// TIA Portal project "Project1" (V19)

(* hardware
DEVICE "S7-1500/ET200MP station_1"  S7-1500 station
   slot 0: "Rail_0"  Rack  6ES7 590-1***0-0AA0
   slot 1: "PLC_1"  CPU 1513-1 PN  6ES7 513-1AL02-0AB0  V2.9
      slot 3: "CPU display_1"  6ES7591-1AA00-0AA0
      slot 32768: "PROFINET interface_1"  X1
         slot 32769: "Port_1"  X1 P1
         slot 32770: "Port_2"  X1 P2
      slot 34817: "Virtual CP interface port_1"  Virtual CP interface port  Virtual CP interface port
   slot 2: "DI 16x24VDC BA_1"  DI 16x24VDC BA  6ES7 521-1BH10-0AA0  V1.1
   slot 3: "DQ 16x24VDC/0.5A BA_1"  DQ 16x24VDC/0.5A BA  6ES7 522-1BH10-0AA0  V1.1
DEVICE "HMI_1"  KTP700 Basic PN
   slot 0: "HMI_1"  KTP700 Basic PN  6AV2 123-2GB03-0AX0  17.0.0.0
   slot 1: "HMI_RT_1"  KTP700 Basic PN  6AV2 123-2GB03-0AX0  17.0.0.0
   slot 5: "HMI_1.IE_CP_1"  PROFINET Interface  17.0.0.0
      slot 1: "PROFINET Interface_1"  PROFINET Interface
         slot 1: "Port_1"  Port
*)

// ===== PLC "PLC_1"  CPU 1513-1 PN =====

VAR_GLOBAL   // PLC tag table "Default tag table"
   "At Entry" AT %I0.0 : Bool;
   "At Load" AT %I0.1 : Bool;
   "At left" AT %I0.2 : Bool;
   "At Middle" AT %I0.3 : Bool;
   "At Right" AT %I0.4 : Bool;
   "At Unload" AT %I0.5 : Bool;
   "At Exit" AT %I0.6 : Bool;
   "Moving X" AT %I0.7 : Bool;
   "Moving Z" AT %I1.0 : Bool;
   "Start" AT %I1.1 : Bool;
   "Reset" AT %I1.2 : Bool;
   "Stop" AT %I1.3 : Bool;
   "Emergency stop" AT %I1.4 : Bool;
   "Auto" AT %I1.5 : Bool;
   "FACTORY I/O (Runing)" AT %I1.6 : Bool;
   "Entry Conveyor" AT %Q0.0 : Bool;
   "Load Conveyor" AT %Q0.1 : Bool;
   "Forks Left" AT %Q0.2 : Bool;
   "Forks Right" AT %Q0.3 : Bool;
   "Lift" AT %Q0.4 : Bool;
   "Unload Conveyor" AT %Q0.5 : Bool;
   "Exit Conveyor" AT %Q0.6 : Bool;
   "Reset light" AT %Q1.0 : Bool;
   "Stop light" AT %Q1.1 : Bool;
   "Target position" AT %QW30 : Int;
   "start light" AT %Q0.7 : Bool;
END_VAR

DATA_BLOCK "GDb"   // DB1
{ S7_Optimized_Access := 'TRUE' }
VERSION : 0.1
   VAR
      "Emergency stop" : Bool;
      Auto : Bool;
      "FACTORY I/O (Runing)" : Bool;
      State0 : Bool := 1;
      State1 : Bool;
      State2 : Bool;
      State3 : Bool;
      State4 : Bool;
      State5 : Bool;
      State6 : Bool;
      State7 : Bool;
      State8 : Bool;
      State9 : Bool;
      t : Int;
      start : Bool;
      stop : Bool;
      startlight : Bool;
      stoplight : Bool;
   END_VAR
BEGIN
END_DATA_BLOCK

// folder: acuators

DATA_BLOCK "acuatorsfb_DB"   // DB2
{ S7_Optimized_Access := 'TRUE' }
VERSION : 0.1
// stored: InstanceOfName acuatorsfb
"acuatorsfb"
BEGIN
END_DATA_BLOCK

// folder: start stop

DATA_BLOCK "startstopdf_DB"   // DB4
{ S7_Optimized_Access := 'TRUE' }
VERSION : 0.1
// stored: InstanceOfName startstopdf
"startstopdf"
BEGIN
END_DATA_BLOCK

// folder: states

DATA_BLOCK "statesfb_DB_1"   // DB3
{ S7_Optimized_Access := 'TRUE' }
VERSION : 0.1
// stored: InstanceOfName statesfb
"statesfb"
BEGIN
END_DATA_BLOCK

// folder: (top level)

ORGANIZATION_BLOCK "Main"   // OB1, LAD, ProgramCycle
TITLE = "Main Program Sweep (Cycle)"
{ S7_Optimized_Access := 'FALSE' }
VERSION : 0.1
   VAR_TEMP
      OB1_EV_CLASS : Byte;   // Bits 0-3 = 1 (Coming event), Bits 4-7 = 1 (Event class 1)
      OB1_SCAN_1 : Byte;   // 1 (Cold restart scan 1 of OB 1), 3 (Scan 2-n of OB 1)
      OB1_PRIORITY : Byte;   // Priority of OB Execution
      OB1_OB_NUMBR : Byte;   // 1 (Organization block 1, OB1)
      OB1_RESERVED_1 : Byte;   // Reserved for system
      OB1_RESERVED_2 : Byte;   // Reserved for system
      OB1_PREV_CYCLE : Int;   // Cycle time of previous OB1 scan (milliseconds)
      OB1_MIN_CYCLE : Int;   // Minimum cycle time of OB1 (milliseconds)
      OB1_MAX_CYCLE : Int;   // Maximum cycle time of OB1 (milliseconds)
      OB1_DATE_TIME : Date_And_Time;   // Date and time OB1 started
   END_VAR
BEGIN

REGION Network 1
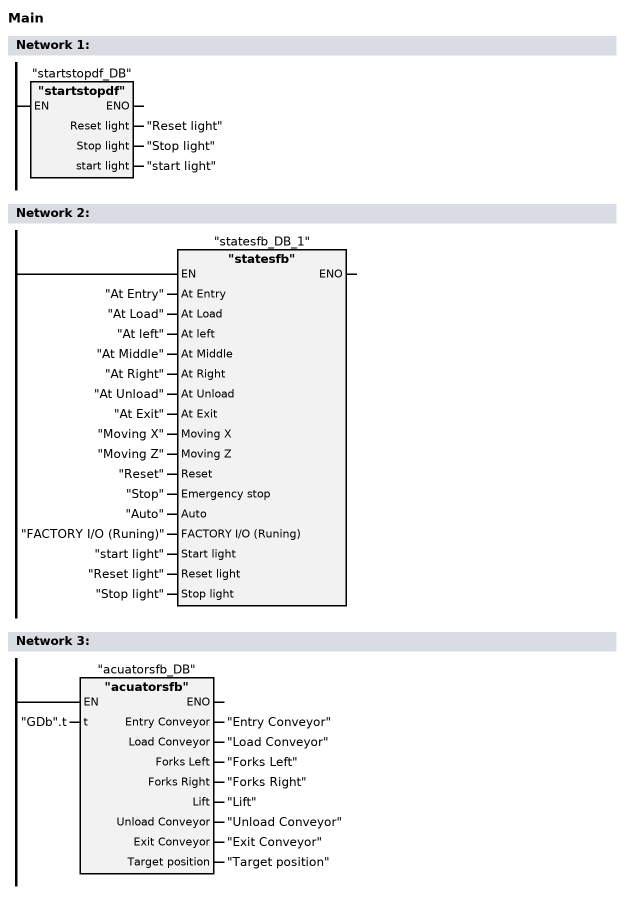
   RUNG wire#powerrail
      "startstopdf_DB"("Reset light" => "Reset light", "Stop light" => "Stop light", "start light" => "start light")
   END_RUNG
   // the same network as SCL:
   "startstopdf_DB"("Reset light" => "Reset light",   // "startstopdf"
                    "Stop light" => "Stop light",
                    "start light" => "start light");
END_REGION

REGION Network 2
   RUNG wire#powerrail
      "statesfb_DB_1"("At Entry" := "At Entry", "At Load" := "At Load", "At left" := "At left", "At Middle" := "At Middle", "At Right" := "At Right", "At Unload" := "At Unload", "At Exit" := "At Exit", "Moving X" := "Moving X", "Moving Z" := "Moving Z", Reset := "Reset", "Emergency stop" := "Stop", Auto := "Auto", "FACTORY I/O (Runing)" := "FACTORY I/O (Runing)", "Start light" := "start light", "Reset light" := "Reset light", "Stop light" := "Stop light")
   END_RUNG
   // the same network as SCL:
   "statesfb_DB_1"("At Entry" := "At Entry",   // "statesfb"
                   "At Load" := "At Load",
                   "At left" := "At left",
                   "At Middle" := "At Middle",
                   "At Right" := "At Right",
                   "At Unload" := "At Unload",
                   "At Exit" := "At Exit",
                   "Moving X" := "Moving X",
                   "Moving Z" := "Moving Z",
                   Reset := "Reset",
                   "Emergency stop" := "Stop",
                   Auto := "Auto",
                   "FACTORY I/O (Runing)" := "FACTORY I/O (Runing)",
                   "Start light" := "start light",
                   "Reset light" := "Reset light",
                   "Stop light" := "Stop light");
END_REGION

REGION Network 3
   RUNG wire#powerrail
      "acuatorsfb_DB"(t := "GDb".t, "Entry Conveyor" => "Entry Conveyor", "Load Conveyor" => "Load Conveyor", "Forks Left" => "Forks Left", "Forks Right" => "Forks Right", Lift => "Lift", "Unload Conveyor" => "Unload Conveyor", "Exit Conveyor" => "Exit Conveyor", "Target position" => "Target position")
   END_RUNG
   // the same network as SCL:
   "acuatorsfb_DB"(t := "GDb".t,   // "acuatorsfb"
                   "Entry Conveyor" => "Entry Conveyor",
                   "Load Conveyor" => "Load Conveyor",
                   "Forks Left" => "Forks Left",
                   "Forks Right" => "Forks Right",
                   Lift => "Lift",
                   "Unload Conveyor" => "Unload Conveyor",
                   "Exit Conveyor" => "Exit Conveyor",
                   "Target position" => "Target position");
END_REGION
END_ORGANIZATION_BLOCK

// folder: acuators

FUNCTION_BLOCK "acuatorsfb"   // FB2, LAD
{ S7_Optimized_Access := 'TRUE' }
VERSION : 0.1
   VAR_OUTPUT
      "Entry Conveyor" : Bool;
      "Load Conveyor" : Bool;
      "Forks Left" : Bool;
      "Forks Right" : Bool;
      Lift : Bool;
      "Unload Conveyor" : Bool;
      "Exit Conveyor" : Bool;
      "Target position" : Int;
   END_VAR
   VAR_IN_OUT
      t : Int;
   END_VAR
   VAR
      Tag_1 : Bool;
      Tag_2 : Bool;
      Tag_3 : Bool;
      Tag_4 : Bool;
      Tag_5 : Bool;
      Tag_6 : Bool;
   END_VAR
   VAR_TEMP   // added for the SCL form of the ladder/FBD networks
      _w1 : Bool;
   END_VAR
BEGIN

REGION Network 2
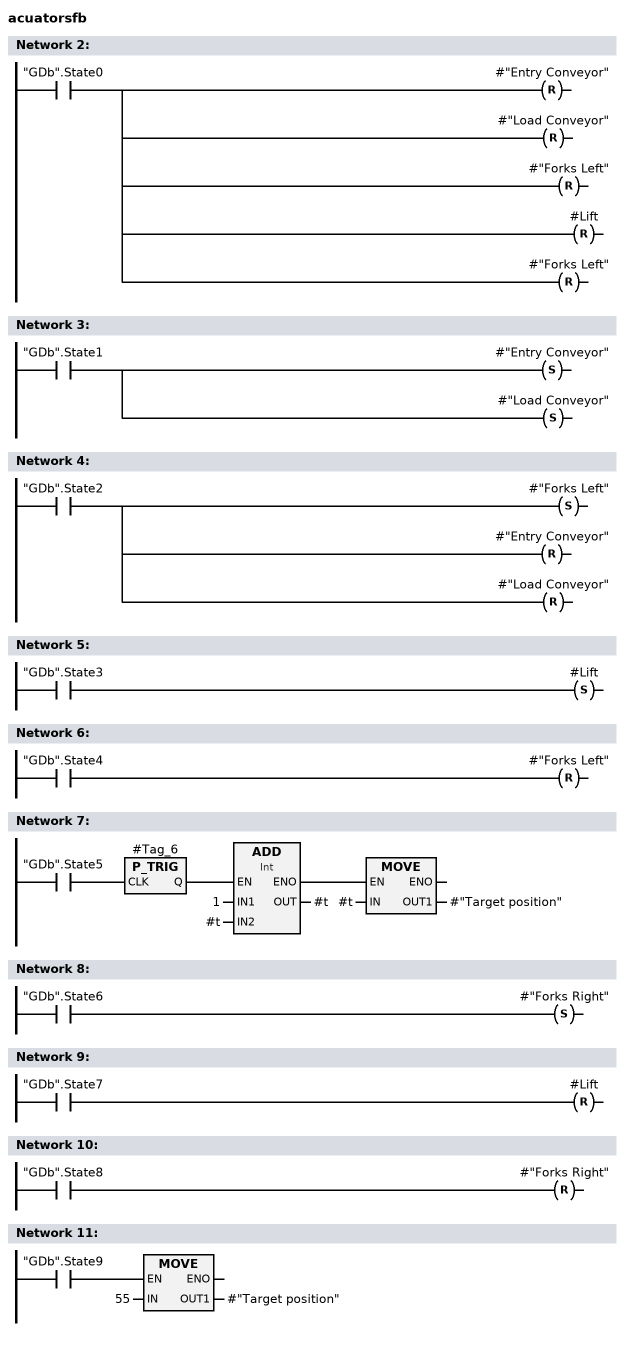
   RUNG wire#powerrail
      Contact( "GDb".State0 )
      wire#w1
      R_Coil( #"Entry Conveyor" )
   END_RUNG
   RUNG wire#w1
      R_Coil( #"Load Conveyor" )
   END_RUNG
   RUNG wire#w1
      R_Coil( #"Forks Left" )
   END_RUNG
   RUNG wire#w1
      R_Coil( #Lift )
   END_RUNG
   RUNG wire#w1
      R_Coil( #"Forks Left" )
   END_RUNG
   // the same network as SCL:
   IF "GDb".State0 THEN
       #"Entry Conveyor" := FALSE;
       #"Load Conveyor" := FALSE;
       #"Forks Left" := FALSE;
       #Lift := FALSE;
       #"Forks Left" := FALSE;
   END_IF;
END_REGION

REGION Network 3
   RUNG wire#powerrail
      Contact( "GDb".State1 )
      wire#w1
      S_Coil( #"Entry Conveyor" )
   END_RUNG
   RUNG wire#w1
      S_Coil( #"Load Conveyor" )
   END_RUNG
   // the same network as SCL:
   IF "GDb".State1 THEN
       #"Entry Conveyor" := TRUE;
       #"Load Conveyor" := TRUE;
   END_IF;
END_REGION

REGION Network 4
   RUNG wire#powerrail
      Contact( "GDb".State2 )
      wire#w1
      S_Coil( #"Forks Left" )
   END_RUNG
   RUNG wire#w1
      R_Coil( #"Entry Conveyor" )
   END_RUNG
   RUNG wire#w1
      R_Coil( #"Load Conveyor" )
   END_RUNG
   // the same network as SCL:
   IF "GDb".State2 THEN
       #"Forks Left" := TRUE;
       #"Entry Conveyor" := FALSE;
       #"Load Conveyor" := FALSE;
   END_IF;
END_REGION

REGION Network 5
   RUNG wire#powerrail
      Contact( "GDb".State3 )
      S_Coil( #Lift )
   END_RUNG
   // the same network as SCL:
   IF "GDb".State3 THEN #Lift := TRUE; END_IF;
END_REGION

REGION Network 6
   RUNG wire#powerrail
      Contact( "GDb".State4 )
      R_Coil( #"Forks Left" )
   END_RUNG
   // the same network as SCL:
   IF "GDb".State4 THEN #"Forks Left" := FALSE; END_IF;
END_REGION

REGION Network 7
   RUNG wire#powerrail
      Contact( "GDb".State5 )
      P_Trig( #Tag_6 )
      { S7_Templates := "SrcType := Int"; S7_GenerateENO := "TRUE" } Add(in1 := 1, in2 := #t, out => #t)
      { S7_GenerateENO := "TRUE" } Move(in := #t, out1 => #"Target position")
   END_RUNG
   // the same network as SCL:
   // ENO of a box is taken as its EN; it also drops when the box reports an error
   #_w1 := "GDb".State5 AND NOT #Tag_6;   // rising edge
   #Tag_6 := "GDb".State5;
   IF #_w1 THEN
       #t := 1 + #t;
       #"Target position" := #t;
   END_IF;
END_REGION

REGION Network 8
   RUNG wire#powerrail
      Contact( "GDb".State6 )
      S_Coil( #"Forks Right" )
   END_RUNG
   // the same network as SCL:
   IF "GDb".State6 THEN #"Forks Right" := TRUE; END_IF;
END_REGION

REGION Network 9
   RUNG wire#powerrail
      Contact( "GDb".State7 )
      R_Coil( #Lift )
   END_RUNG
   // the same network as SCL:
   IF "GDb".State7 THEN #Lift := FALSE; END_IF;
END_REGION

REGION Network 10
   RUNG wire#powerrail
      Contact( "GDb".State8 )
      R_Coil( #"Forks Right" )
   END_RUNG
   // the same network as SCL:
   IF "GDb".State8 THEN #"Forks Right" := FALSE; END_IF;
END_REGION

REGION Network 11
   RUNG wire#powerrail
      Contact( "GDb".State9 )
      { S7_GenerateENO := "TRUE" } Move(in := 55, out1 => #"Target position")
   END_RUNG
   // the same network as SCL:
   IF "GDb".State9 THEN #"Target position" := 55; END_IF;
END_REGION
END_FUNCTION_BLOCK

// folder: start stop

FUNCTION_BLOCK "startstopdf"   // FB3, LAD
{ S7_Optimized_Access := 'TRUE' }
VERSION : 0.1
   VAR_OUTPUT
      "Reset light" : Bool;
      "Stop light" : Bool;
      "start light" : Bool;
   END_VAR
BEGIN

REGION Network 2
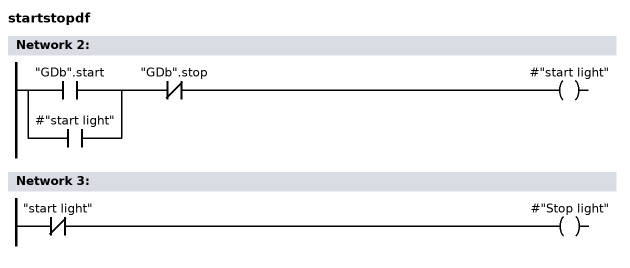
   RUNG wire#powerrail
      Contact( "GDb".start )
      wire#w1
      I_Contact( "GDb".stop )
      Coil( #"start light" )
   END_RUNG
   RUNG wire#powerrail
      Contact( #"start light" )
   END_RUNG wire#w1
   // the same network as SCL:
   #"start light" := ("GDb".start OR #"start light") AND NOT "GDb".stop;
END_REGION

REGION Network 3
   RUNG wire#powerrail
      I_Contact( "start light" )
      Coil( #"Stop light" )
   END_RUNG
   // the same network as SCL:
   #"Stop light" := NOT "start light";
END_REGION
END_FUNCTION_BLOCK

// folder: states

FUNCTION_BLOCK "statesfb"   // FB1, LAD
{ S7_Optimized_Access := 'TRUE' }
VERSION : 0.1
   VAR_INPUT
      "At Entry" : Bool;
      "At Load" : Bool;
      "At left" : Bool;
      "At Middle" : Bool;
      "At Right" : Bool;
      "At Unload" : Bool;
      "At Exit" : Bool;
      "Moving X" : Bool;
      "Moving Z" : Bool;
      Reset : Bool;
      "Emergency stop" : Bool;
      Auto : Bool;
      "FACTORY I/O (Runing)" : Bool;
      "Start light" : Bool;
      "Reset light" : Bool;
      "Stop light" : Bool;
   END_VAR
   VAR
      Tag_1 : Bool;
      Tag_2 : Bool;
      Tag_3 : Bool;
      Tag_4 : Bool;
      Tag_5 : Bool;
   END_VAR
   VAR_TEMP   // added for the SCL form of the ladder/FBD networks
      _w1 : Bool;
      _w2 : Bool;
   END_VAR
BEGIN

REGION Network 1
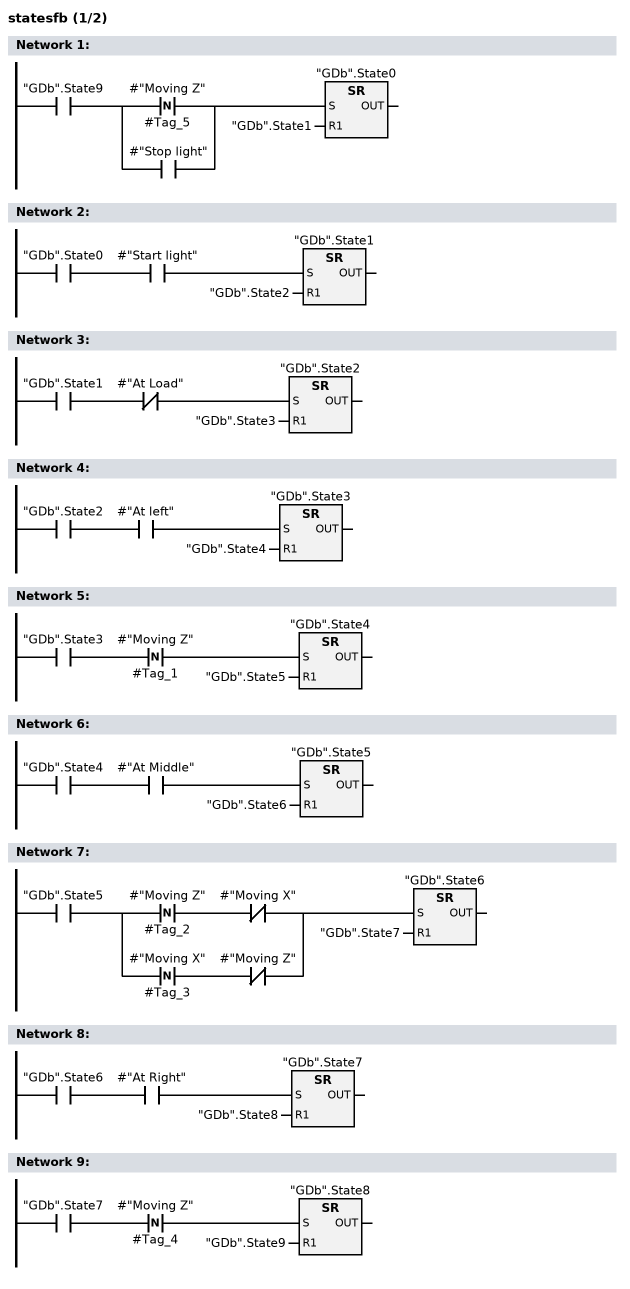
   RUNG wire#powerrail
      Contact( "GDb".State9 )
      wire#w1
      N_Contact(operand := #"Moving Z", bit := #Tag_5)
      wire#w2
      S_SR(operand := "GDb".State0, r1 := "GDb".State1)
   END_RUNG
   RUNG wire#w1
      Contact( #"Stop light" )
   END_RUNG wire#w2
   // the same network as SCL:
   #_w1 := "GDb".State9 AND NOT #"Moving Z" AND #Tag_5;   // falling edge of #"Moving Z"
   #Tag_5 := #"Moving Z";
   IF #_w1 OR ("GDb".State9 AND #"Stop light") THEN
       "GDb".State0 := TRUE;   // SR flip-flop
   END_IF;
   IF "GDb".State1 THEN "GDb".State0 := FALSE; END_IF;
END_REGION

REGION Network 2
   RUNG wire#powerrail
      Contact( "GDb".State0 )
      Contact( #"Start light" )
      S_SR(operand := "GDb".State1, r1 := "GDb".State2)
   END_RUNG
   // the same network as SCL:
   IF "GDb".State0 AND #"Start light" THEN
       "GDb".State1 := TRUE;   // SR flip-flop
   END_IF;
   IF "GDb".State2 THEN "GDb".State1 := FALSE; END_IF;
END_REGION

REGION Network 3
   RUNG wire#powerrail
      Contact( "GDb".State1 )
      I_Contact( #"At Load" )
      S_SR(operand := "GDb".State2, r1 := "GDb".State3)
   END_RUNG
   // the same network as SCL:
   IF "GDb".State1 AND NOT #"At Load" THEN
       "GDb".State2 := TRUE;   // SR flip-flop
   END_IF;
   IF "GDb".State3 THEN "GDb".State2 := FALSE; END_IF;
END_REGION

REGION Network 4
   RUNG wire#powerrail
      Contact( "GDb".State2 )
      Contact( #"At left" )
      S_SR(operand := "GDb".State3, r1 := "GDb".State4)
   END_RUNG
   // the same network as SCL:
   IF "GDb".State2 AND #"At left" THEN
       "GDb".State3 := TRUE;   // SR flip-flop
   END_IF;
   IF "GDb".State4 THEN "GDb".State3 := FALSE; END_IF;
END_REGION

REGION Network 5
   RUNG wire#powerrail
      Contact( "GDb".State3 )
      N_Contact(operand := #"Moving Z", bit := #Tag_1)
      S_SR(operand := "GDb".State4, r1 := "GDb".State5)
   END_RUNG
   // the same network as SCL:
   #_w1 := "GDb".State3 AND NOT #"Moving Z" AND #Tag_1;   // falling edge of #"Moving Z"
   #Tag_1 := #"Moving Z";
   IF #_w1 THEN
       "GDb".State4 := TRUE;   // SR flip-flop
   END_IF;
   IF "GDb".State5 THEN "GDb".State4 := FALSE; END_IF;
END_REGION

REGION Network 6
   RUNG wire#powerrail
      Contact( "GDb".State4 )
      Contact( #"At Middle" )
      S_SR(operand := "GDb".State5, r1 := "GDb".State6)
   END_RUNG
   // the same network as SCL:
   IF "GDb".State4 AND #"At Middle" THEN
       "GDb".State5 := TRUE;   // SR flip-flop
   END_IF;
   IF "GDb".State6 THEN "GDb".State5 := FALSE; END_IF;
END_REGION

REGION Network 7
   RUNG wire#powerrail
      Contact( "GDb".State5 )
      wire#w1
      N_Contact(operand := #"Moving Z", bit := #Tag_2)
      I_Contact( #"Moving X" )
      wire#w2
      S_SR(operand := "GDb".State6, r1 := "GDb".State7)
   END_RUNG
   RUNG wire#w1
      N_Contact(operand := #"Moving X", bit := #Tag_3)
      I_Contact( #"Moving Z" )
   END_RUNG wire#w2
   // the same network as SCL:
   #_w1 := "GDb".State5 AND NOT #"Moving Z" AND #Tag_2;   // falling edge of #"Moving Z"
   #Tag_2 := #"Moving Z";
   #_w2 := "GDb".State5 AND NOT #"Moving X" AND #Tag_3;   // falling edge of #"Moving X"
   #Tag_3 := #"Moving X";
   IF (#_w1 AND NOT #"Moving X") OR (#_w2 AND NOT #"Moving Z") THEN
       "GDb".State6 := TRUE;   // SR flip-flop
   END_IF;
   IF "GDb".State7 THEN "GDb".State6 := FALSE; END_IF;
END_REGION

REGION Network 8
   RUNG wire#powerrail
      Contact( "GDb".State6 )
      Contact( #"At Right" )
      S_SR(operand := "GDb".State7, r1 := "GDb".State8)
   END_RUNG
   // the same network as SCL:
   IF "GDb".State6 AND #"At Right" THEN
       "GDb".State7 := TRUE;   // SR flip-flop
   END_IF;
   IF "GDb".State8 THEN "GDb".State7 := FALSE; END_IF;
END_REGION

REGION Network 9
   RUNG wire#powerrail
      Contact( "GDb".State7 )
      N_Contact(operand := #"Moving Z", bit := #Tag_4)
      S_SR(operand := "GDb".State8, r1 := "GDb".State9)
   END_RUNG
   // the same network as SCL:
   #_w1 := "GDb".State7 AND NOT #"Moving Z" AND #Tag_4;   // falling edge of #"Moving Z"
   #Tag_4 := #"Moving Z";
   IF #_w1 THEN
       "GDb".State8 := TRUE;   // SR flip-flop
   END_IF;
   IF "GDb".State9 THEN "GDb".State8 := FALSE; END_IF;
END_REGION

REGION Network 10
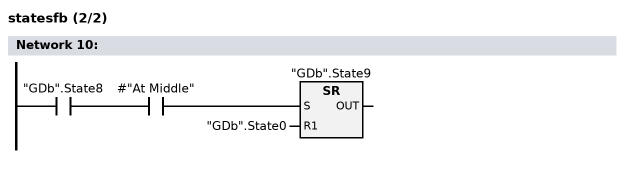
   RUNG wire#powerrail
      Contact( "GDb".State8 )
      Contact( #"At Middle" )
      S_SR(operand := "GDb".State9, r1 := "GDb".State0)
   END_RUNG
   // the same network as SCL:
   IF "GDb".State8 AND #"At Middle" THEN
       "GDb".State9 := TRUE;   // SR flip-flop
   END_IF;
   IF "GDb".State0 THEN "GDb".State9 := FALSE; END_IF;
END_REGION
END_FUNCTION_BLOCK

(* ===== HMI "HMI_RT_1" =====
system functions are stored by id; their names below are inferred from use
connection "HMI_Connection_1": ETHERNET, SMART_S7_1500_OMS

HMI tags "Default tag table"
   "Tag_ScreenNumber" : UInt, internal
   "Start light" : Bool = PLC "start light" AT %Q0.7, 1 s
   "Start" : Bool = PLC Start AT %I1.1, 1 s
   "Stop" : Bool = PLC Stop AT %I1.3, 1 s
   "t" : Int = PLC GDb.t AT %QW30, 1 s
   "GDb_start" : Bool = PLC GDb.start, 1 s
   "GDb_stop" : Bool = PLC GDb.stop, 1 s
   "GDb_startlight" : Bool = PLC GDb.startlight, 1 s
   "GDb_t" : Int = PLC GDb.t, 1 s
   "Target position" : Int = PLC "Target position" AT %QW30, 1 s

Template "Template_1" 800x480
   Button "Exit" at 714,429 size 71x50; TextOff 'Exit'; PictureOff "ExitRuntime_KTP700_Basic_PN_TR"; PictureOn "ExitRuntime_KTP700_Basic_PN_TR"
      on Release: StopRuntime(0)
   Button "Template_Button" at 614,429 size 71x50; TextOff 'Text'
   Button "Template_Button_1" at 514,429 size 71x50; TextOff 'Text'
   Button "Template_Button_2" at 414,429 size 71x50; TextOff 'Text'
   Button "Template_Button_3" at 314,429 size 71x50; TextOff 'Text'
   Button "Template_Button_4" at 214,429 size 71x50; TextOff 'Text'
   Button "Alarms" at 114,429 size 71x50; TextOff 'Alarms'; PictureOff "AlarmDisplay_KTP700_Basic_PN_TR"; PictureOn "AlarmDisplay_KTP700_Basic_PN_TR"
      on Release: function_ef3f5d25("Alarm window_Unacknowledged", -1)
   Button "Start screen" at 14,429 size 71x50; TextOff 'Start screen'; PictureOff "NavigateHome_KTP700_Basic_PN_TR"; PictureOn "NavigateHome_KTP700_Basic_PN_TR"
      on Release: ActivateScreen("Root screen", 0)
   SymbolicIOField "Symbolic_IO_Field_Screen" at 93,9 size 600x33; TextOff '0'; TextOn '1'; TextList "TextList_ScreenNames"
      ProcessValue <- "Tag_ScreenNumber"
      on Change: ActivateScreenByNumber("Tag_ScreenNumber", 0)
   DateTimeField "HmiScreenItemData" at 695,25 size 105x25
   DateTimeField "HmiScreenItemData_1" at 695,0 size 105x25
   GraphicView "Logo" at 0,0 size 91x51; Picture "Logo of HMI_1"

screen "Root screen" 800x480, template "Template_1"
   on GenerateScreen: SetTag("Tag_ScreenNumber", 1)
   TextField "HmiScreenItemData" at 80,225 size 640x25; Text 'Automated Warehouse'
   Button "Button_2" at 423,274 size 192x32; TextOff 'Automatic'; TextOn 'Screen_1'
      on Click: ActivateScreen("Screen_1", 0)
   Button "Button_3" at 182,274 size 192x32; TextOff 'Manual'; TextOn 'Screen_1'

screen "Screen_1" 800x480
   Button "Button_1" at 206,168 size 96x32; TextOff 'Start'
      on Click: SetBit("GDb_start"); ResetBit("GDb_stop")
   Button "Button_2" at 206,257 size 96x32; TextOff 'Stop'
      on Click: SetBit("GDb_stop"); ResetBit("GDb_start")
   Rectangle "Rectangle_1" at 422,168 size 96x48
      Appearance <- "Start light"
   IOField "I/O field_1" at 422,257 size 94x77; FormatPattern 999
      ProcessValue <- "GDb_t"
   Button "Button_3" at 1,445 size 192x32; TextOff 'Root screen'
      on Click: ActivateScreen("Root screen", 0)
*)